TYPE (* IEC 61131-3,Table 12#5 *)
  (* Standard: 61131-3; Type: Data Type; Description: Table 12, #5 *)
  (* Version 0.0, 2000-11-09, JHC, Rockwell Automation *)
  (* Compiler header: package fb.rt.ita; *)
  (* Compiler Java IBM VisualAge 3.0 *)
  (* ASN.1 tag PRIVATE 16 *)
  FILTER_PARAMETER : SINT(0..99);
END_TYPE
